(*********************************** G.D S.p.A. - Technical Department ***********************************
============= PROGRAM INFO ============
FOLDER:             TBD
MACHINES INVOLVED:  TBD 

============= DESCRIPTION =============
csp main interface program

============= REVISIONS ===============
Date		Version	 	Author      	Description             
----------	-------		------------  	--------------------------------------------
2019/09/27 	0000.00	 	M.Grasso		Creation of the PRG

**********************************************************************************************************)
PROGRAM _csp_main_lowest
VAR
END_VAR

(*MAIN*)
	
	(*Drives*)
	
	(*Motorization*)
	
	(*Cam Manager*)
	
	(*Services*)
	
	(*Interface*)
	
	(*Safety*)
	;

END_PROGRAM

(* stored: Version 1.1.0.1, ProductVersion 3.1.4022.12
   POU _csp_main_lowest: Id {96ff0a3e-71bd-4284-9bf0-e3e01da0d2b4}, SpecialFunc None *)
